Staubli VAL3: Refresh.pgx

program Refresh()
begin
  //
  if bUserRefresh
    cls()
    userPage()
    gotoxy(1,1)
    put("F1->选中路径转换")
    gotoxy(1,13)
    put("转换")
    gotoxy(1,2)
    put("F2->全部转换")
    gotoxy(6,13)
    put("全部")
    gotoxy(1,3)
    put("F3->删除路径")
    gotoxy(11,13)
    put("删除")
//    gotoxy(1,4)
//    put("F4->")
//    gotoxy(16,13)
//    put("")
    //
//    gotoxy(1,6)
//    put("F6->")
//    gotoxy(26,13)
//    put("")
//    gotoxy(1,7)
//    put("F7->")
//    gotoxy(31,13)
//    put("")
    gotoxy(1,7)
    put("F8->返回")
    gotoxy(36,13)
    put("返回")
  endIf
end
